SUBAPPLICATION Softkey_Aux_Switch_TO_Remote_WRITE_BG_OPC (* VT-SoftKey lesen ODER AUX-Zuweisung (Joystick) lesen ODER lokaler Web-Override ODER physischer Remote-Taster auf einem dritten Modul + Remote-OPC-UA-Write an Zielmodul + VT-Hintergrundfarbe (SoftKey UND AUX) aus Remote-Subscribe (4-Quellen-Variante von Softkey_Aux_IXA_TO_Remote_WRITE_BG_OPC, fuer Funktionen mit einem zusaetzlichen fest verbauten Taster auf einem dritten Modul, z.B. Schnittverstellung) *)
  (* Standard: 61499-2; Description: Copyright (c) 2026 Meisterschulen am Ostbahnhof This program and the accompanying materials are made available under the terms of the Eclipse Public License 2.0 which is available at https://www.eclipse.org/legal/epl-2.0/ SPDX-License-Identifier: EPL-2.0 *)
  (* Version 1.0, 2026-09-07, Franz Höpfinger, Meisterschulen am Ostbahnhof, initial API and implementation and/or initial documentation - 4-Quellen-Variante fuer Schnittverstellung (V14) *)
  PACKAGE MyLib::sys;
  (* Documentation:
  SoftKey UND Aux UND Web UND Remote-Taster → Remote-OPC-UA-Write mit Status-Feedback (ein Kanal)
   Duennwandiger Wrapper, der Softkey_Aux_Switch_TO_Remote_WRITE (Kommando: 4 Quellen → Remote-Write) und AX_SUBSCRIBE_BG3_WEB_OPC (Status: Remote-Subscribe → Hintergrundfarbe auf SoftKey UND Aux + lokaler Web-Republish, unveraendert von der Standard-3-Quellen-Variante wiederverwendet) nebeneinanderstellt.
   Fuer den Standardfall (3 Quellen: SoftKey/AUX/Web, kein zusaetzlicher Taster auf einem dritten Modul) weiterhin Softkey_Aux_IXA_TO_Remote_WRITE_BG_OPC verwenden.
  *)
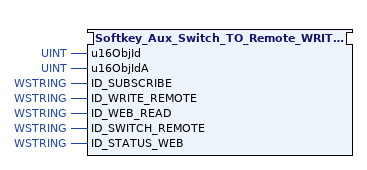
  VAR_INPUT
    u16ObjId : UINT; (* Object ID SoftKey/Hintergrund (VT) *)
    u16ObjIdA : UINT; (* Object ID AuxFunction2/Hintergrund (VT) *)
    ID_SUBSCRIBE : WSTRING; (* Remote-Subscribe-Adresse (Status/Farbe, ACTION=SUBSCRIBE) *)
    ID_WRITE_REMOTE : WSTRING; (* Remote-Write-Adresse zum Zielmodul (Befehl, ACTION=WRITE, CLIENT) *)
    ID_WEB_READ : WSTRING; (* Lokale Subscribe-Adresse fuer einen Web-Client (z.B. vt-ui-mirror) auf demselben Modul, ODER-verknuepft mit SoftKey und AUX *)
    ID_SWITCH_REMOTE : WSTRING; (* Remote-Subscribe-Adresse eines zusaetzlichen physischen Tasters auf einem ANDEREN Modul, ODER-verknuepft mit SoftKey/AUX/Web *)
    ID_STATUS_WEB : WSTRING; (* Lokale Publish-Adresse (auf diesem Modul) fuer den vom Zielmodul zurueckgemeldeten Zustand - damit ein Web-Client (z.B. vt-ui-mirror) dieselbe Hintergrundfarbe wie das echte VT zeigen kann *)
  END_VAR
  SUBAPPS
    Command : MyLib::sys::Softkey_Aux_Switch_TO_Remote_WRITE;
    Status : MyLib::sys::AX_SUBSCRIBE_BG3_WEB_OPC;
  END_SUBAPPS
  DATA_CONNECTIONS
    u16ObjId TO Command.u16ObjId;
    u16ObjIdA TO Command.u16ObjIdA;
    ID_WRITE_REMOTE TO Command.ID_WRITE_REMOTE;
    ID_WEB_READ TO Command.ID_WEB_READ;
    ID_SWITCH_REMOTE TO Command.ID_SWITCH_REMOTE;
    u16ObjId TO Status.u16ObjId;
    u16ObjIdA TO Status.u16ObjIdA;
    ID_SUBSCRIBE TO Status.ID_SUBSCRIBE;
    ID_STATUS_WEB TO Status.ID_STATUS_WEB;
  END_CONNECTIONS
END_SUBAPPLICATION
